# EPICS substitutions: ioc_tops/ioc_bpm/BPMApp/Db/user.substitutions
# Example substitutions file

file "db/circle.db" {
    { user = "scs" }
}

file "db/dbExample1.db" {
    { user = "scs" }
}

file db/dbExample2.db {
    pattern { user, no, scan }
        { "scs", 1, "1 second" }
        { "scs", 2, "2 second" }
        { "scs", 3, "5 second" }
}
